TYPE DUT_COORD_REF :
STRUCT
    X, Y, Z, A, B, C: LREAL;
END_STRUCT
END_TYPE

(* stored: Version 1.1.0.1
   DUT DUT_COORD_REF: Id {37a476e8-8045-4532-a808-d8c44ae7a0c4} *)
